// TIA Portal V17 export
// export: Created 2023-04-03T06:31:40.7323767Z, ExportSetting WithDefaults, DisplayName Totally Integrated Automation Portal, DisplayVersion V17 Update 4, DisplayName TIA Portal Openness, DisplayVersion V17 Update 4, DisplayName TIA Portal Version Control Interface, DisplayVersion V17, DisplayName STEP 7 Professional, DisplayVersion V17 Update 4, DisplayName STEP 7 Safety, DisplayVersion V17, DisplayName WinCC Professional, DisplayVersion V17 Update 4
DATA_BLOCK "clock"   // DB4
{ S7_Optimized_Access := 'TRUE' }
VERSION : 0.1
// stored: AutoNumber true, DBAccessibleFromOPCUA true, DBAccessibleFromWebserver true, IsOnlyStoredInLoadMemory false, IsRetainMemResEnabled false, IsWriteProtectedInAS false, MemoryReserve 100
   VAR
      xClock_5Hz : Bool;
      xClock_2_5Hz : Bool;
      xClock_2Hz : Bool;
      xClock_1_25Hz : Bool;
      xClock_1Hz : Bool;
      xClock_0_625Hz : Bool;
      xClock_0_5Hz : Bool;
      xClock_10Hz : Bool;
   END_VAR
BEGIN
END_DATA_BLOCK
